FUNCTION_BLOCK EscritaAnalogica (* Basic Function Block Type *)
  (* Standard: 61499-2 *)
  (* Version 0.0, 02/03/2026, Template *)
  PACKAGE Hidryco.HidrycoLib;
  EC_STATES
    START; (* Initial State *)
  END_STATES
  ALGORITHM INIT IN ST: (* Initialization algorithm *)
;
  END_ALGORITHM
  ALGORITHM REQ IN ST: (* Normally executed algorithm *)
;
  END_ALGORITHM
END_FUNCTION_BLOCK
